{attribute 'qualified_only'}
VAR_GLOBAL	
	extrusionWeight : REAL;
	
	extrusionHeight : REAL;
	extrusionWidth : REAL;
END_VAR

(* stored: Version 1.1.0.1, ProductVersion 3.1.4024.11
   GVL ExtrusionData: Id {367ca7b9-1246-46ec-b5c0-6c54f2fc7615} *)
